Fanuc KAREL source: ks00003.KL

-- PROVISIONAL review KL for V940-1; original PC SHA256 aa7c9fec62f15ac3fb55e2c0a41cd22f0a8a8ffd8300ff14a3a0b304b80ec890
-- Incomplete behavior may be omitted. Consult companion uncertainty JSON. Do not deploy.
PROGRAM KS00003
%NOLOCKGROUP
VAR
  FLAG : BOOLEAN
  N : INTEGER
  STATUS : INTEGER
  PN : STRING[80]
  VN : STRING[80]
-- UNRESOLVED_DECL A type=001100
-- UNRESOLVED_DECL B type=001100
BEGIN
  -- V9_ZERO_TABLE_METADATA_HINT layout=0001; no indexed target words; source/name/runtime held
  -- UNRESOLVED_PC offsets 5-13; opcodes 3F,75
  -- UNRESOLVED_PC offsets 18-27; opcodes 3F,75
  -- UNRESOLVED_PC offsets 32-47; opcodes 22,22,30
  -- UNRESOLVED_PC offsets 52-56; opcodes 7F
END KS00003
